// TIA Portal project "modbus_master" (V15.1)

(* hardware
DEVICE "S7-1200 station_1"  S7-1200 Station
   slot 0: "Rack_0"  S7-1200 Rack  Rack  V1.0
   slot 1: "PLC_1"  CPU 1214C DC/DC/DC  6ES7 214-1AG40-0XB0  V4.2
*)

// ===== PLC "PLC_1"  CPU 1214C DC/DC/DC =====

VAR_GLOBAL   // PLC tag table "默认变量表"
   "Tag_1" AT %I0.0 : Bool;
   "Tag_2" AT %Q0.0 : Bool;
   "Tag_3" AT %I0.1 : Bool;
   "Tag_4" AT %M10.0 : Bool;
   "Tag_5" AT %M10.1 : Bool;
   "Tag_6" AT %M10.2 : Bool;
   "Tag_7" AT %MW12 : Word;
   "Rec_REQ" AT %M2.0 : Bool;
   "Rec_DONE" AT %M2.1 : Bool;
   "Rec_BUSY" AT %M2.2 : Bool;
   "Rec_ERROR" AT %M2.3 : Bool;
   "Send_REQ" AT %M2.4 : Bool;
   "Send_DONE" AT %M2.5 : Bool;
   "Send_BUSY" AT %M2.6 : Bool;
   "Send_ERROR" AT %M2.7 : Bool;
   "Rec_STATUS" AT %MW4 : Word;
   "Rec_ERRORCODE" AT %MW6 : Word;
   "Send_STATUS" AT %MW8 : Word;
   "Send_ERRORCODE" AT %MW10 : Word;
   "Tag_8" AT %M0.0 : Bool;
   "System_Byte" AT %MB1 : Byte;
   "FirstScan" AT %M1.0 : Bool;
   "DiagStatusUpdate" AT %M1.1 : Bool;
   "AlwaysTRUE" AT %M1.2 : Bool;
   "AlwaysFALSE" AT %M1.3 : Bool;
   "Clock_Byte" AT %MB0 : Byte;
   "Clock_10Hz" AT %M0.0 : Bool;
   "Clock_5Hz" AT %M0.1 : Bool;
   "Clock_2.5Hz" AT %M0.2 : Bool;
   "Clock_2Hz" AT %M0.3 : Bool;
   "Clock_1.25Hz" AT %M0.4 : Bool;
   "Clock_1Hz" AT %M0.5 : Bool;
   "Clock_0.625Hz" AT %M0.6 : Bool;
   "Clock_0.5Hz" AT %M0.7 : Bool;
END_VAR

DATA_BLOCK "Connect"   // DB1
{ S7_Optimized_Access := 'TRUE' }
VERSION : 0.1
   VAR
      modbus_rt : TCON_IP_v4;
   END_VAR
BEGIN
   modbus_rt.InterfaceId := 64;
   modbus_rt.ID := 1;
   modbus_rt.ConnectionType := 11;
   modbus_rt.ActiveEstablished := 1;
   modbus_rt.RemoteAddress.ADDR[1] := 192;
   modbus_rt.RemoteAddress.ADDR[2] := 168;
   modbus_rt.RemoteAddress.ADDR[3] := 28;
   modbus_rt.RemoteAddress.ADDR[4] := 254;
   modbus_rt.RemotePort := 502;
   modbus_rt.LocalPort := 0;
END_DATA_BLOCK

DATA_BLOCK "Data_Modbus"   // DB8
{ S7_Optimized_Access := 'FALSE' }
VERSION : 0.1
   VAR
      Recive : Array[0..14] of Bool;
      Send : Array[0..9] of Bool;
   END_VAR
BEGIN
END_DATA_BLOCK

ORGANIZATION_BLOCK "Main"   // OB1, LAD, ProgramCycle
TITLE = "Main Program Sweep (Cycle)"
{ S7_Optimized_Access := 'TRUE' }
VERSION : 0.1
   VAR_INPUT
      Initial_Call : Bool;   // Initial call of this OB
      Remanence : Bool;   // =True, if remanent data are available
   END_VAR
BEGIN

REGION Network 1: 启动modbus
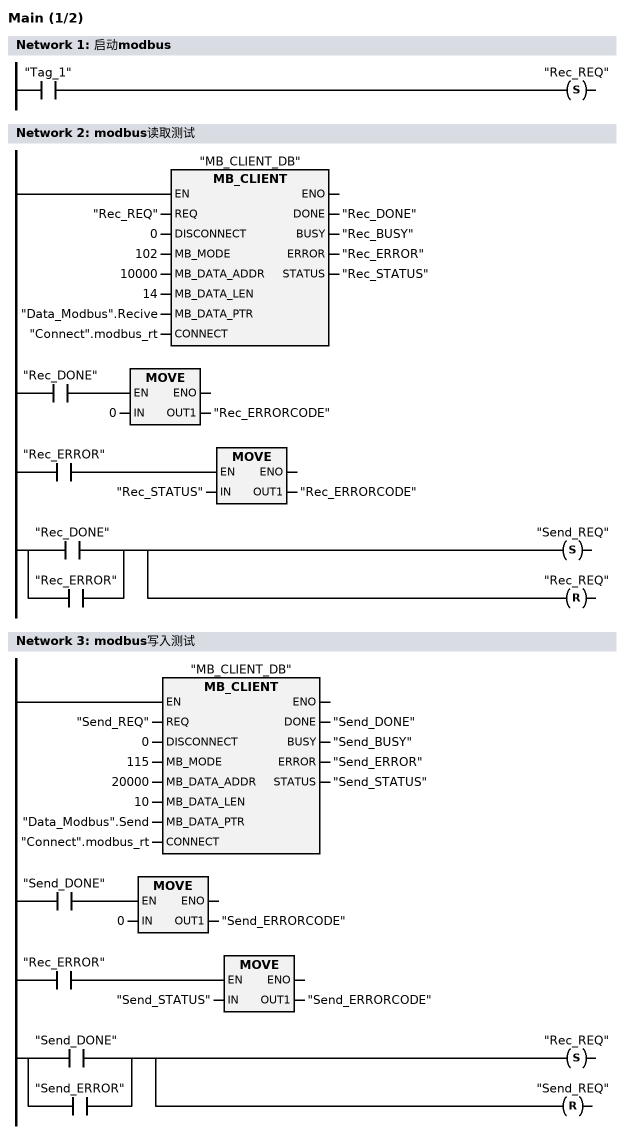
   RUNG wire#powerrail
      Contact( "Tag_1" )
      S_Coil( "Rec_REQ" )
   END_RUNG
   // the same network as SCL:
   IF "Tag_1" THEN "Rec_REQ" := TRUE; END_IF;
END_REGION

REGION Network 2: modbus读取测试
   "MB_CLIENT_DB"(REQ := "Rec_REQ",   // MB_CLIENT
                  DISCONNECT := 0,
                  MB_MODE := 102,
                  MB_DATA_ADDR := 10000,
                  MB_DATA_LEN := 14,
                  MB_DATA_PTR := "Data_Modbus".Recive,
                  CONNECT := "Connect".modbus_rt,
                  DONE => "Rec_DONE",
                  BUSY => "Rec_BUSY",
                  ERROR => "Rec_ERROR",
                  STATUS => "Rec_STATUS");
   IF "Rec_DONE" THEN "Rec_ERRORCODE" := 0; END_IF;
   IF "Rec_ERROR" THEN "Rec_ERRORCODE" := "Rec_STATUS"; END_IF;
   IF "Rec_DONE" OR "Rec_ERROR" THEN
       "Send_REQ" := TRUE;
       "Rec_REQ" := FALSE;
   END_IF;
END_REGION

REGION Network 3: modbus写入测试
   "MB_CLIENT_DB"(REQ := "Send_REQ",   // MB_CLIENT
                  DISCONNECT := 0,
                  MB_MODE := 115,
                  MB_DATA_ADDR := 20000,
                  MB_DATA_LEN := 10,
                  MB_DATA_PTR := "Data_Modbus".Send,
                  CONNECT := "Connect".modbus_rt,
                  DONE => "Send_DONE",
                  BUSY => "Send_BUSY",
                  ERROR => "Send_ERROR",
                  STATUS => "Send_STATUS");
   IF "Send_DONE" THEN "Send_ERRORCODE" := 0; END_IF;
   IF "Rec_ERROR" THEN "Send_ERRORCODE" := "Send_STATUS"; END_IF;
   IF "Send_DONE" OR "Send_ERROR" THEN
       "Rec_REQ" := TRUE;
       "Send_REQ" := FALSE;
   END_IF;
END_REGION

REGION Network 4: 同步输入信号到输出信号上
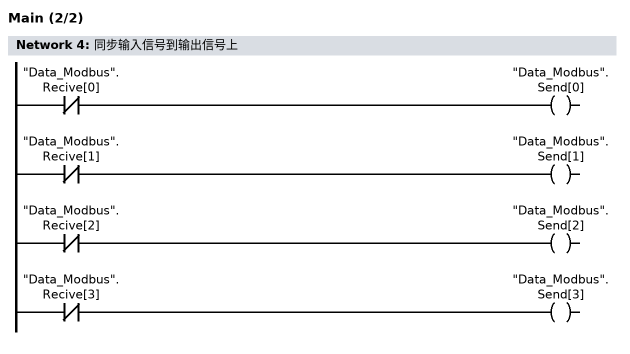
   RUNG wire#powerrail
      I_Contact( "Data_Modbus".Recive[0] )
      Coil( "Data_Modbus".Send[0] )
   END_RUNG
   RUNG wire#powerrail
      I_Contact( "Data_Modbus".Recive[1] )
      Coil( "Data_Modbus".Send[1] )
   END_RUNG
   RUNG wire#powerrail
      I_Contact( "Data_Modbus".Recive[2] )
      Coil( "Data_Modbus".Send[2] )
   END_RUNG
   RUNG wire#powerrail
      I_Contact( "Data_Modbus".Recive[3] )
      Coil( "Data_Modbus".Send[3] )
   END_RUNG
   // the same network as SCL:
   "Data_Modbus".Send[0] := NOT "Data_Modbus".Recive[0];
   "Data_Modbus".Send[1] := NOT "Data_Modbus".Recive[1];
   "Data_Modbus".Send[2] := NOT "Data_Modbus".Recive[2];
   "Data_Modbus".Send[3] := NOT "Data_Modbus".Recive[3];
END_REGION
END_ORGANIZATION_BLOCK